// TwinCAT 3 PLC project PLC01
// ProgramVersion: 3.1.4023.0
// libraries:
//   Tc2_Standard, * (Beckhoff Automation GmbH)
//   Tc2_System, * (Beckhoff Automation GmbH)
//   Tc2_Utilities, * (Beckhoff Automation GmbH)
//   Tc3_Database, * (Beckhoff Automation GmbH)
//   Tc3_EventLogger, * (Beckhoff Automation GmbH)
//   Tc3_Module, * (Beckhoff Automation GmbH)
// project tree:
//   DUTs/ E_ORDERTYPE.TcDUT, ST_Record.TcDUT
//   GVLs/ GVL.TcGVL
//   / PlcTask.TcTTO
//   POUs/ MAIN.TcPOU, pReadDB.TcPOU, pWriteDB.TcPOU
// real-time tasks:
//   TASK PlcTask: cycle T#10ms, priority 20, ADS port 350

CONFIGURATION PLC01
    RESOURCE PLC ON TwinCAT3
        TASK PlcTask(INTERVAL := T#10ms, PRIORITY := 20);
        PROGRAM MAIN WITH PlcTask : MAIN;
    END_RESOURCE
END_CONFIGURATION

// ---- DUTs/E_ORDERTYPE.TcDUT

{attribute 'qualified_only'}
TYPE E_ORDERTYPE :
(
    ASC := 0,
    DESC := 1
);
END_TYPE

// ---- DUTs/ST_Record.TcDUT
TYPE ST_Record :
STRUCT
	ID: LINT;
	Timestamp: DT;
	Name: STRING(80);
	nSensor1: LREAL;
	nSensor2: LREAL;
END_STRUCT
END_TYPE

// ---- GVLs/GVL.TcGVL
{attribute 'qualified_only'}
VAR_GLOBAL
fbPLCDBRead    	: FB_PLCDBReadEvt (sNetID := '', tTimeout := T#5S);
fbPLCDBWrite    :  FB_PLCDBWriteEvt(sNetID := '', tTimeout := T#5S);
END_VAR

// ---- POUs/MAIN.TcPOU
PROGRAM MAIN
VAR

	nState: INT;

END_VAR


(*Setup a database  -  In that database make a table using this command in the Sql Query Editor...

CREATE TABLE `MyTable_Struct` 
(
	`ID` BIGINT NOT NULL AUTO_INCREMENT, 
	 `Timestamp` DATETIME, 
	 `Name` VARCHAR(80), 
	 `nSensor1` DOUBLE, 
	 `nSensor2` DOUBLE,

	 PRIMARY KEY (ID)
)

*)

CASE nState OF
	
0: //Idle

1: //DB write
	pWriteDB();
	IF NOT GVL.fbPLCDBWrite.bBusy THEN
		
		IF NOT GVL.fbPLCDBWrite.bError THEN
			nState := 2;
			ELSE
			nState := 3;
		END_IF;
	END_IF
	
2: //DB read
	pReadDB();
	IF NOT GVL.fbPLCDBRead.bBusy  THEN

		IF NOT GVL.fbPLCDBRead.bError THEN
			nState := 0;
			ELSE
			nState := 3;
		END_IF;
	END_IF;
	
3: //Error state


END_CASE

END_PROGRAM

// ---- POUs/pWriteDB.TcPOU
PROGRAM pWriteDB
VAR
	//fbPLCDBWrite    :  FB_PLCDBWriteEvt(sNetID := '', tTimeout := T#5S);
    myRecord        :  ST_Record;
    ColumnNames     :  ARRAY[0..4] OF STRING(50);
    
    systime         :  GETSYSTEMTIME;
    currentTime     :  T_FILETIME;
    tcMessage       :  I_TcMessage;
	
	nState			: INT;
	
	nSensor1		: LREAL;
	nSensor2		: LREAL;
	
END_VAR

// set Values
systime(timeLoDw => currentTime.dwLowDateTime, timeHiDW => currentTime.dwHighDateTime );
myRecord.Timestamp := FILETIME_TO_DT(currentTime);
myRecord.Name       := 'MyStructVal';
myRecord.nSensor1    := nSensor1;
myRecord.nSensor2    := nSensor2;

// set columnnames
ColumnNames[0] := 'ID';
ColumnNames[1] := 'Timestamp';
ColumnNames[2] := 'Name';
ColumnNames[3] := 'nSensor1';
ColumnNames[4] := 'nSensor2';

// Call Functionblock
IF GVL.fbPLCDBWrite.WriteStruct(
    hDBID:= 1, 
    sTableName:= 'myTable_Struct', 
    pRecord:= ADR(myRecord), 
    cbRecord:= SIZEOF(myRecord), 
    pColumnNames:= ADR(ColumnNames) , 
    cbColumnNames:= SIZEOF(ColumnNames))
THEN
    IF GVL.fbPLCDBWrite.bError THEN
        tcMessage := GVL.fbPLCDBWrite.ipTcResult;
        nState := 255; 
    ELSE
        nState := 0;
    END_IF
END_IF

METHOD WriteStruct : BOOL
VAR_INPUT
	hDBID: UDINT;
    sTableName: T_MaxString;
    pRecord: POINTER TO BYTE;
    cbRecord: UDINT;
    pColumnNames: POINTER TO ARRAY [0..MAX_DBCOLUMNS] OF STRING(50);
    cbColumnNames: UDINT;
END_VAR
END_METHOD

END_PROGRAM

// ---- POUs/pReadDB.TcPOU
PROGRAM pReadDB
VAR
	//fbPLCDBRead    	: FB_PLCDBReadEvt (sNetID := '', tTimeout := T#5S);
    myCustomStruct 	: ST_Record; //where the data will be stored
    tcMessage      	: I_TcMessage; 
	nState			: INT;
	ColumnNames 	: ARRAY [0..4] OF STRING(50); //table column names.
END_VAR

//Reads a struct from database.

// set columnnames
ColumnNames[0] := 'ID';
ColumnNames[1] := 'Timestamp';
ColumnNames[2] := 'Name';
ColumnNames[3] := 'nSensor1';
ColumnNames[4] := 'nSensor2';

IF GVL.fbPLCDBRead.ReadStruct(
    hDBID:= 1, 
    sTableName:= 'MyTable_Struct', //name of the table to read from.
    pColumnNames:= ADR(ColumnNames), 
    cbColumnNames:= SIZEOF(ColumnNames), 
    sOrderByColumn:= ColumnNames[0], 
    eOrderType:= E_OrderType.ASC, 
    nStartIndex:= 3, //get the data corresponding to ID 3 in the database. 
    nRecordCount:= 1, //how many records to get.
    pData:= ADR(myCustomStruct), 
    cbData:= SIZEOF(myCustomStruct))
THEN
    IF GVL.fbPLCDBRead.bError THEN
        tcMessage:= GVL.fbPLCDBRead.ipTcResult;
        nState := 255; 
    ELSE
        nState := 0;
    END_IF
END_IF


//

METHOD ReadStruct : BOOL
VAR_INPUT
   hDBID: UDINT;
    sTableName: T_MaxString;
    pColumnNames: POINTER TO ARRAY [0..MAX_DBCOLUMNS] OF STRING(50);
    cbColumnNames: UDINT;
    sOrderByColumn: STRING(50);
  //  eOrderType: E_OrderType := E_OrderType.eOrder_ASC;
  	eOrderType : E_OrderType := E_OrderType.ASC;
    nStartIndex: UDINT;
    nRecordCount: UDINT;
    pData: POINTER TO BYTE;
    cbData: UDINT;
END_VAR
END_METHOD

END_PROGRAM
